Yaskawa INFORM job: MOTOTAC1.JBI

/JOB
//NAME MOTOTAC1
///FOLDERNAME INNE
//POS
///NPOS 11,11,0,0,0,0
///TOOL 0
///POSTYPE PULSE
///PULSE
C00000=32571,-80067,-84751,-11816,58952,90735
C00001=31607,89434,-37773,-14900,117198,84049
C00002=27942,106739,-15544,-12222,112315,84109
C00003=27775,104829,-15576,-12051,111361,84188
C00004=27737,105172,-15154,-12022,111277,84191
C00005=27775,104829,-15576,-12051,111361,84188
C00006=27942,106739,-15544,-12222,112315,84109
C00007=34849,33621,-59846,-28051,60630,87205
C00008=33063,35985,-55736,-26897,59113,87161
C00009=45284,24434,-87718,-33795,73184,85659
C00010=32571,-80067,-84751,-11816,58952,90735
BC00000=204899,1734,820586
BC00001=204899,578,1075157
BC00002=204899,578,1075155
BC00003=204899,578,1075157
BC00004=204899,578,1075157
BC00005=204899,578,1075157
BC00006=204899,578,1075155
BC00007=204899,578,1075157
BC00008=204899,578,1075157
BC00009=204899,578,1075157
BC00010=204899,1734,820586
//INST
///DATE 2024/02/06 15:42
///ATTR SC,RW
///GROUP1 RB1,BS1
///LVARS 20,10,20,3,10,26,26,0
NOP
*TOP
COMM PAUSE IF IN#(1563)=OFF
'---------SET MODE 0=RUN 1=ADJUST
SET LB010 0
'------------------------SET TOOL
SET LB011 0
'----------------SET DIRECT INPUT
SET LB012 1
'-------------SET WIREFEED OUTPUT
SET LD013 4095
'---------------SET WIREFEED TIME
SET LI000 80
'-------------SET WIRE CUT OUTPUT
SET LD014 16
'-------SET AIR CLEAN BLOW OUTPUT
SET LD015 4091
'----------------SET LIMITS IN mm
SET LD004 5
'--------------------------------
'-----------PREPARING LP VARIABLE
MUL LD004 1000
SET LD000 1
*1
GETS LPX[LD000] $PX000
CNVRT LPX[LD000] LPX[LD000] RF
SUB LP[LD000] LP[LD000]
ADD LD000 1
JUMP *1 IF LD000<21
PAUSE IF LB010=1
'WRITE TOOL ORIGINAL DATA HERE
SETE LP010 (1) -48546
SETE LP010 (2) -907
SETE LP010 (3) 608610
SETE LP010 (4) 1800000
SETE LP010 (5) -220000
SETE LP010 (6) 0
JUMP *RUN1 IF LB010=1
*WRITE
PAUSE IF LB010=1
'----WRITE IN STOP POS. DATA HERE
SETE LP019 (1) 1844713
SETE LP019 (2) -527591
SETE LP019 (3) -85073
SETE LP019 (4) 80751
SETE LP019 (5) -643669
SETE LP019 (6) -94866
JUMP *END IF LB010=1
'------PREPARE DIALOG BOX--------
JUMP *RUN1 IF LB010=1
GETE LD000 LP010 (4)
GETE LD001 LP010 (5)
GETE LD002 LP010 (6)
SET LB000 0
SET LB001 1
SET LB002 2
SET LB003 4
SET LB004 5
SET LB005 7
SET LB006 12
SET LB007 3
SET LS000 "TOOLDAT_IS_OUT.."
SET LS001 "OFF_LIMIT.."
SET LS002 "CONTINUE/STOP.."
SET LS003 "CONTINUE"
SET LS004 " STOP."
SET LS005 "CHECK/CHANGE.."
SET LS006 " TOOL.THEN.."
SET LS007 " RUN_THIS_JOB.."
SET LS009 "FROM_BEGINNING.."
SET LS008 "....OK...."
JUMP *RUN4
*RUN1
SET LB000 0
SET LB001 1
SET LB002 2
SET LB003 4
SET LB004 7
SET LS000 "READ_CURR.POS.."
SET LS001 "IN_ROBOT_COORD.."
SET LS002 "NAME_IT_STOP.."
SET LS004 "OK"
JUMP *RUN
*RUN2
CNVRT LPX008 LPX008 RF
CNVRT LPX009 LPX009 RF
ADD LP008 LP009
DIV LP008 2
MOVL LP008 V=33.3 PL=0
SET LP011 LP008
MSHIFT LPX015 TF LPX019 LPX011
SET LP017 LP010
INVMAT LP012 LP011
MULMAT LP013 LP017 LP012
MULMAT LP018 LP013 LP019
SETE LP018 (4) LD000
SETE LP018 (5) LD001
SETE LP018 (6) LD002
SETTOOL TL#(LB011) LP018
'----------------------------TOOL
SUB LP010 LP018
GETE LD000 LP010 (1)
GETE LD001 LP010 (2)
GETE LD002 LP010 (3)
SET I070 LD000
SET I071 LD001
SET I072 LD002
DIV I070 -100
DIV I071 -100
DIV I072 -100
JUMP *TOOL-ERR IF LD000>LD004
JUMP *TOOL-ERR IF LD001>LD004
JUMP *TOOL-ERR IF LD002>LD004
DIV LD004 -1
JUMP *TOOL-ERR IF LD000<=LD004
JUMP *TOOL-ERR IF LD001<=LD004
JUMP *TOOL-ERR IF LD002<=LD004
JUMP *OK
*TOOL-ERR
DIALOG B030 DIALSB LB000 LB000 LS000 LB000 LB004 LS003 DIALSB LB000 LB001 LS001 LB006 LB004 LS004 DIALSB LB000 LB002 LS002
JUMP *OK IF B030<>2
DIALOG B030 DIALSB LB000 LB000 LS005 LB004 LB004 LS008 DIALSB LB000 LB001 LS006 DIALSB LB000 LB002 LS007 DIALSB LB000 LB007 LS009
PAUSE
JUMP *TOP
*OK
JUMP *END
*RUN3
ADD LP008 LP009
DIV LP008 2
MOVL LP008 V=50.0
DIALOG B030 DIALSB LB000 LB000 LS000 LB004 LB003 LS004 DIALSB LB000 LB001 LS001 DIALSB LB000 LB002 LS002
JUMP *WRITE
*RUN
'----------CHECKING TOOL POSITION
JUMP *RUN5 IF LB010=1
*RUN4
SETTOOL TL#(LB011) LP010
*RUN5
SETE LP001 (3) -25000
SETE LP002 (3) 5000
SETE LP003 (1) 50000
SETE LP004 (1) -50000
SETE LP005 (2) 50000
SETE LP006 (2) -50000
SETE LP007 (1) -5000
'------------------START POSITION
PAUSE IF LB010=1
'POS. FROM HOME TO WIRECUT UNIT
'AND TO CUP
MOVJ C00000 BC00000 VJ=50.00
MOVJ C00001 BC00001 VJ=50.00
MOVJ C00002 BC00002 VJ=50.00
PULSE OT#(LD013) T=LI000
MOVL C00003 BC00003 V=75.0
MOVL C00004 BC00004 V=16.7
TIMER T=0.30
DOUT OT#(LD014) ON
TIMER T=1.00
MOVL C00005 BC00005 V=50.0
DOUT OT#(LD014) OFF
MOVL C00006 BC00006 V=100.0
MOVL C00007 BC00007 V=750.0
MOVJ C00008 BC00008 VJ=25.00 PL=0
PULSE OT#(LD015) T=1.00
WAIT SOUT#(394)=OFF
IMOV LP001 V=10.8 PL=0 TF SRCH RIN#(LB012)=ON T=0.30 DIS=50.0
IMOV LP002 V=33.3 PL=0 TF
TIMER T=0.20
WAIT SOUT#(394)=OFF
IMOV LP003 V=10.8 PL=0 TF SRCH RIN#(LB012)=ON T=0.30 DIS=10.0
GETS LPX008 $PX001
IMOV LP007 V=33.3 PL=0 TF
TIMER T=0.20
WAIT SOUT#(394)=OFF
IMOV LP004 V=10.8 PL=0 TF SRCH RIN#(LB012)=ON T=0.30 DIS=10.0
GETS LPX009 $PX001
ADD LP008 LP009
DIV LP008 2
MOVL LP008 V=66.7
TIMER T=0.20
WAIT SOUT#(394)=OFF
IMOV LP005 V=10.8 PL=0 TF SRCH RIN#(LB012)=ON T=0.30 DIS=10.0
GETS LPX009 $PX001
MOVL LP008 V=66.7
TIMER T=0.20
WAIT SOUT#(394)=OFF
IMOV LP006 V=10.8 PL=0 TF SRCH RIN#(LB012)=ON T=0.30 DIS=10.0
GETS LPX008 $PX001
JUMP *RUN2 IF LB010=0
JUMP *RUN3 IF LB010=1
PAUSE
*END
PAUSE IF LB010=1
'POSITIONS FROM CUP TO HOME
MOVJ C00009 BC00009 VJ=25.00
MOVJ C00010 BC00010 VJ=50.00
END
